// TIA Portal project "FactoryIO_Template_S7-1200_V16_V16" (V16)
// Vorlageprojekt für das Buch mit Zielsystem S7-1200

(* hardware
DEVICE "S7-1200-Station_1"  S7-1200 Station
   slot 0: "Baugruppenträger_0"  Rack  V1.0
   slot 1: "PLC_1"  CPU 1211C DC/DC/DC  6ES7 211-1AE40-0XB0  V4.1
*)

// ===== PLC "PLC_1"  CPU 1211C DC/DC/DC =====

VAR_GLOBAL   // PLC tag table "Standard-Variablentabelle"
   "belt_conv_0" AT %A0.0 : Bool;
   "start" AT %E0.0 : Bool;
   "stop" AT %E0.1 : Bool;
   "Tag_4" AT %I10.0 : Bool;
   "Tag_5" AT %Q10.0 : Bool;
   "Tag_6" AT %I10.1 : Bool;
   "run marker" AT %M0.0 : Bool;
   "stop load" AT %M0.4 : Bool;
   "Tag_3" AT %M6.1 : Bool;
   "belt_conv_0_Marker" AT %M5.0 : Bool;
   "Expect_off_Marker" AT %M1.7 : Bool;
   "run load" AT %M0.3 : Bool;
   "load_AC_marker" AT %M5.1 : Bool;
   "At_0_sens" AT %I0.5 : Bool;
   "mid_sens_Box" AT %I0.3 : Bool;
   "large_sens_Box" AT %I0.4 : Bool;
   "large_sens_marker" AT %M1.5 : Bool;
   "Tag_2" AT %M2.0 : Bool;
   "Expect_sens_marker" AT %M1.6 : Bool;
   "elevator_right_limit" AT %I1.2 : Bool;
   "Tag_7" AT %M0.2 : Bool;
   "Out_at_1_sens 11" AT %M1.0 : Bool;
   "At 2 High_sens _marker" AT %M2.4 : Bool;
   "Save_marker_Down" AT %M5.7 : Bool;
   "Save marker up" AT %M5.2 : Bool;
   "At_1_low_sens" AT %I0.6 : Bool;
   "Tag_8" AT %M0.5 : Bool;
   "out_at_1 sens" AT %M0.6 : Bool;
   "Slow_marker" AT %M5.3 : Bool;
   "At_low_sens_positive 2_marker" AT %M2.2 : Bool;
   "At_high_sens 1" AT %I0.7 : Bool;
   "Tag_9" AT %M0.7 : Bool;
   "Entry_1_Neg_marker" AT %M1.4 : Bool;
   "Entry_2_neg_marker" AT %M4.3 : Bool;
   "unload_marker" AT %M5.4 : Bool;
   "Entry_conv_1" AT %I1.3 : Bool;
   "Tag_10" AT %M1.1 : Bool;
   "entry_1_+_marker" AT %M1.2 : Bool;
   "Tag_11" AT %M1.3 : Bool;
   "belt_conv_1_marker" AT %M5.5 : Bool;
   "at_low_sens 2" AT %I1.0 : Bool;
   "Tag_12" AT %M2.1 : Bool;
   "at 2 high sens" AT %I1.1 : Bool;
   "Tag_13" AT %M2.3 : Bool;
   "entry_conv_2" AT %I1.4 : Bool;
   "Tag_14" AT %M4.2 : Bool;
   "Entry_2_+_marker" AT %M4.0 : Bool;
   "belt_conv_2_marker" AT %M5.6 : Bool;
   "load_Ac" AT %Q0.3 : Bool;
   "up" AT %Q0.5 : Bool;
   "slow" AT %Q0.7 : Bool;
   "unload" AT %Q0.4 : Bool;
   "belt_conv_1" AT %Q0.1 : Bool;
   "belt_conv_2" AT %Q0.2 : Bool;
   "down" AT %Q0.6 : Bool;
   "Tag_1" AT %M4.1 : Bool;
END_VAR

FUNCTION "MHJ-PLC-Lab-Function-S71200" : Void   // FC9000, SCL
{ S7_Optimized_Access := 'TRUE' }
VERSION : 0.1
   VAR_TEMP
      rdTimeReturn : Int;
      outputTime : DTL;
      SyncVal : Byte;
      forVal : Int;
      forVal_2 : Int;
      Value : Byte;
   END_VAR
   VAR CONSTANT
      CompVal : Byte := 16#34;
      Value_01 : Byte := 16#11;
      Value_01_DW : DWord := 16#A165_D992;
      Value_02_DW : DWord := 16#58BE_4401;
   END_VAR
BEGIN

   #Value:=PEEK(area := 16#82,
        dbNumber := 0,
        byteOffset := 511);
   #Value := #Value + 1;

   POKE(area := 16#82,
        dbNumber := 0,
        byteOffset := 511,
        value := #Value);

   POKE(area:=16#81,
        dbNumber:=0,
        byteOffset:=1016,
        value:=#Value_01_DW);
   POKE(area := 16#81,
        dbNumber := 0,
        byteOffset := 1020,
        value := #Value_02_DW);

   POKE(area := 16#81,
        dbNumber := 0,
        byteOffset := 511,
        value := B#16#00);

   FOR #forVal := 0 TO 120 DO
       FOR #forVal_2:=0 TO 10 DO
           #rdTimeReturn:=RD_SYS_T(#outputTime);
           #rdTimeReturn := WR_SYS_T(#outputTime);
           #rdTimeReturn := RD_SYS_T(#outputTime);
           #rdTimeReturn := WR_SYS_T(#outputTime);
       END_FOR;
       #SyncVal:= PEEK(area := 16#81,
                      dbNumber := 0,
                      byteOffset := 511);
       IF #SyncVal = #CompVal THEN
          GOTO M_1;
       END_IF;
   END_FOR;
   RETURN;

   M_1:
   POKE(area := 16#81,
        dbNumber := 0,
        byteOffset := 511,
        value := B#16#0);
END_FUNCTION

ORGANIZATION_BLOCK "Main"   // OB1, LAD, ProgramCycle
TITLE = "Main Program Sweep (Cycle)"
{ S7_Optimized_Access := 'TRUE' }
VERSION : 0.1
   VAR_INPUT
      Initial_Call : Bool;   // Initial call of this OB
      Remanence : Bool;   // =True, if remanent data are available
   END_VAR
   VAR_TEMP   // added for the SCL form of the ladder/FBD networks
      _w1 : Bool;
      _w2 : Bool;
      _w3 : Bool;
      _w4 : Bool;
      _w5 : Bool;
      _w6 : Bool;
      _w7 : Bool;
      _w8 : Bool;
      _w9 : Bool;
      _w10 : Bool;
   END_VAR
BEGIN

REGION Network 1: Konnektierungsbaustein für PLC-Lab
   // Im Netzwerk 1 wird der Konnektierungsbaustein für PLC-Lab aufgerufen.
   // Dieser Aufruf darf nicht entfernt werden!
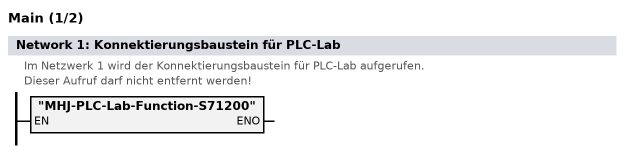
   RUNG wire#powerrail
      "MHJ-PLC-Lab-Function-S71200"()
   END_RUNG
   // the same network as SCL:
   "MHJ-PLC-Lab-Function-S71200"();
END_REGION

REGION Network 2
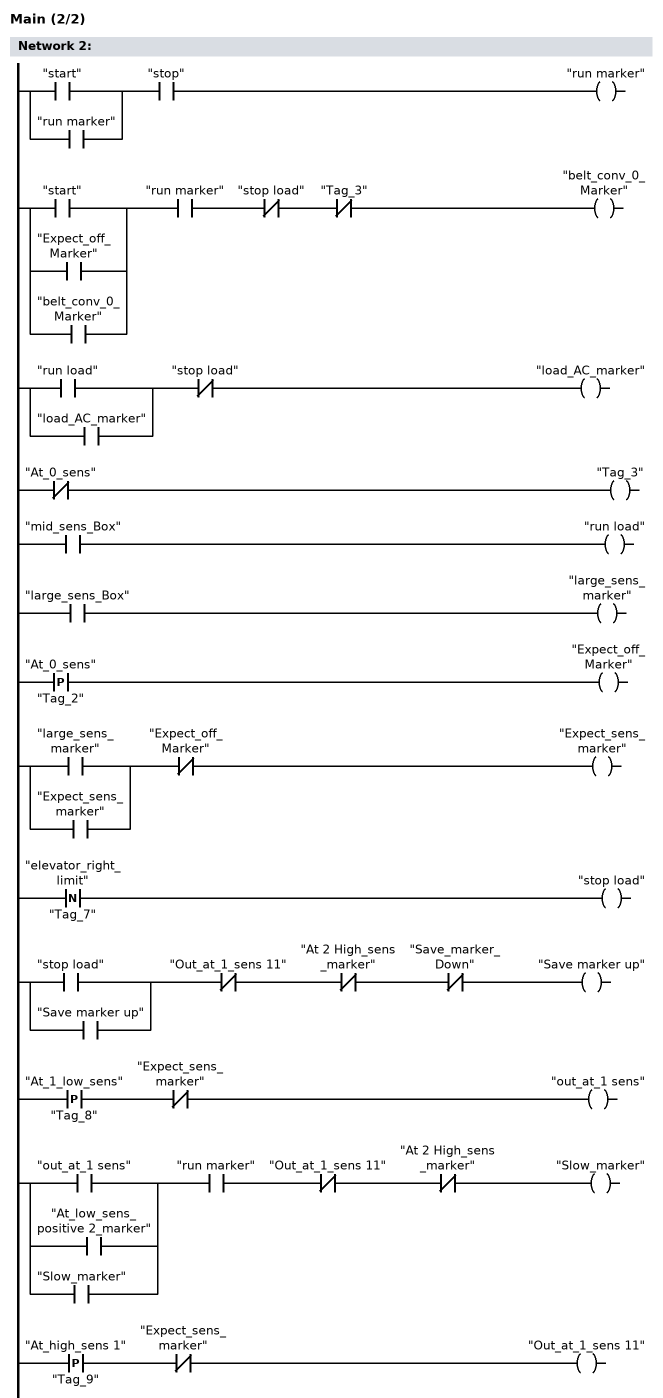
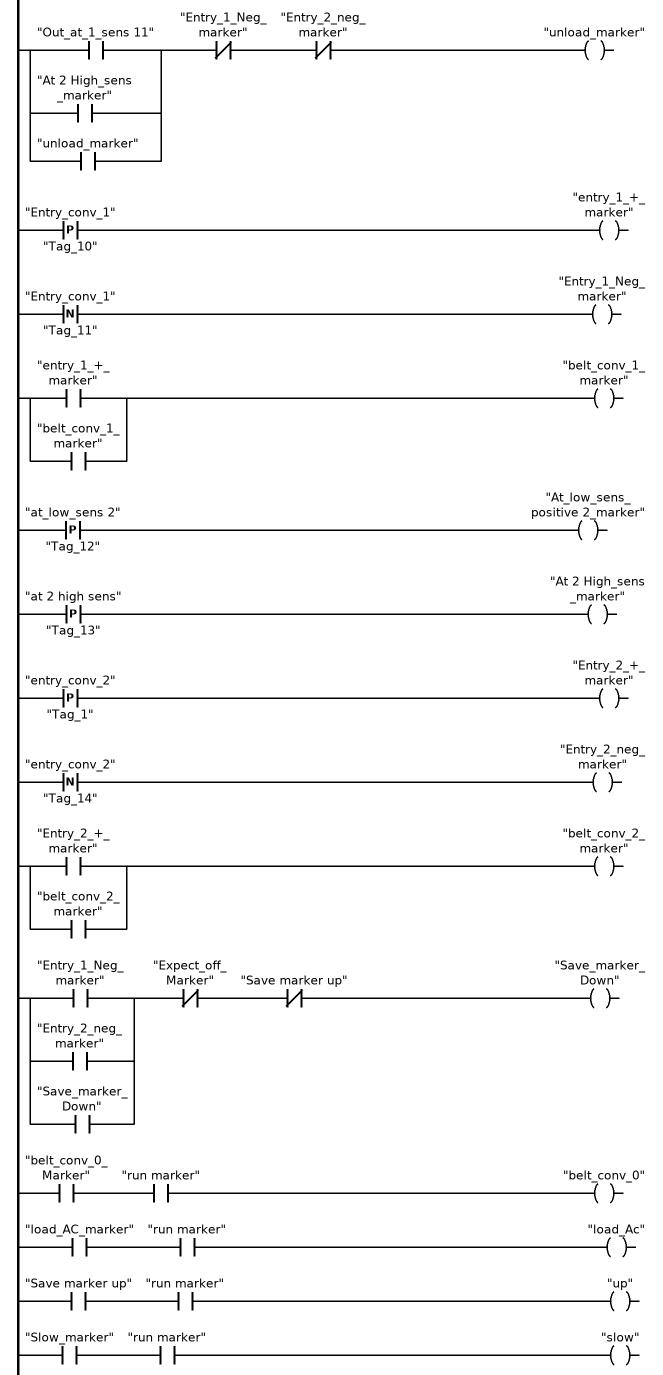
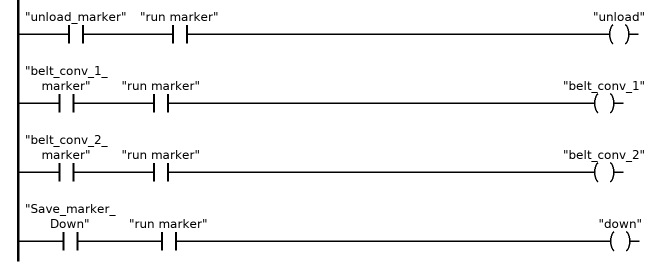
   RUNG wire#powerrail
      Contact( "start" )
      wire#w1
      Contact( "stop" )
      Coil( "run marker" )
   END_RUNG
   RUNG wire#powerrail
      Contact( "run marker" )
   END_RUNG wire#w1
   RUNG wire#powerrail
      Contact( "start" )
      wire#w2
      Contact( "run marker" )
      I_Contact( "stop load" )
      I_Contact( "Tag_3" )
      Coil( "belt_conv_0_Marker" )
   END_RUNG
   RUNG wire#powerrail
      Contact( "Expect_off_Marker" )
   END_RUNG wire#w2
   RUNG wire#powerrail
      Contact( "belt_conv_0_Marker" )
   END_RUNG wire#w2
   RUNG wire#powerrail
      Contact( "run load" )
      wire#w3
      I_Contact( "stop load" )
      Coil( "load_AC_marker" )
   END_RUNG
   RUNG wire#powerrail
      Contact( "load_AC_marker" )
   END_RUNG wire#w3
   RUNG wire#powerrail
      I_Contact( "At_0_sens" )
      Coil( "Tag_3" )
   END_RUNG
   RUNG wire#powerrail
      Contact( "mid_sens_Box" )
      Coil( "run load" )
   END_RUNG
   RUNG wire#powerrail
      Contact( "large_sens_Box" )
      Coil( "large_sens_marker" )
   END_RUNG
   RUNG wire#powerrail
      P_Contact(operand := "At_0_sens", bit := "Tag_2")
      Coil( "Expect_off_Marker" )
   END_RUNG
   RUNG wire#powerrail
      Contact( "large_sens_marker" )
      wire#w4
      I_Contact( "Expect_off_Marker" )
      Coil( "Expect_sens_marker" )
   END_RUNG
   RUNG wire#powerrail
      Contact( "Expect_sens_marker" )
   END_RUNG wire#w4
   RUNG wire#powerrail
      N_Contact(operand := "elevator_right_limit", bit := "Tag_7")
      Coil( "stop load" )
   END_RUNG
   RUNG wire#powerrail
      Contact( "stop load" )
      wire#w5
      I_Contact( "Out_at_1_sens 11" )
      I_Contact( "At 2 High_sens _marker" )
      I_Contact( "Save_marker_Down" )
      Coil( "Save marker up" )
   END_RUNG
   RUNG wire#powerrail
      Contact( "Save marker up" )
   END_RUNG wire#w5
   RUNG wire#powerrail
      P_Contact(operand := "At_1_low_sens", bit := "Tag_8")
      I_Contact( "Expect_sens_marker" )
      Coil( "out_at_1 sens" )
   END_RUNG
   RUNG wire#powerrail
      Contact( "out_at_1 sens" )
      wire#w6
      Contact( "run marker" )
      I_Contact( "Out_at_1_sens 11" )
      I_Contact( "At 2 High_sens _marker" )
      Coil( "Slow_marker" )
   END_RUNG
   RUNG wire#powerrail
      Contact( "At_low_sens_positive 2_marker" )
   END_RUNG wire#w6
   RUNG wire#powerrail
      Contact( "Slow_marker" )
   END_RUNG wire#w6
   RUNG wire#powerrail
      P_Contact(operand := "At_high_sens 1", bit := "Tag_9")
      I_Contact( "Expect_sens_marker" )
      Coil( "Out_at_1_sens 11" )
   END_RUNG
   RUNG wire#powerrail
      Contact( "Out_at_1_sens 11" )
      wire#w7
      I_Contact( "Entry_1_Neg_marker" )
      I_Contact( "Entry_2_neg_marker" )
      Coil( "unload_marker" )
   END_RUNG
   RUNG wire#powerrail
      Contact( "At 2 High_sens _marker" )
   END_RUNG wire#w7
   RUNG wire#powerrail
      Contact( "unload_marker" )
   END_RUNG wire#w7
   RUNG wire#powerrail
      P_Contact(operand := "Entry_conv_1", bit := "Tag_10")
      Coil( "entry_1_+_marker" )
   END_RUNG
   RUNG wire#powerrail
      N_Contact(operand := "Entry_conv_1", bit := "Tag_11")
      Coil( "Entry_1_Neg_marker" )
   END_RUNG
   RUNG wire#powerrail
      Contact( "entry_1_+_marker" )
      wire#w8
      Coil( "belt_conv_1_marker" )
   END_RUNG
   RUNG wire#powerrail
      Contact( "belt_conv_1_marker" )
   END_RUNG wire#w8
   RUNG wire#powerrail
      P_Contact(operand := "at_low_sens 2", bit := "Tag_12")
      Coil( "At_low_sens_positive 2_marker" )
   END_RUNG
   RUNG wire#powerrail
      P_Contact(operand := "at 2 high sens", bit := "Tag_13")
      Coil( "At 2 High_sens _marker" )
   END_RUNG
   RUNG wire#powerrail
      P_Contact(operand := "entry_conv_2", bit := "Tag_1")
      Coil( "Entry_2_+_marker" )
   END_RUNG
   RUNG wire#powerrail
      N_Contact(operand := "entry_conv_2", bit := "Tag_14")
      Coil( "Entry_2_neg_marker" )
   END_RUNG
   RUNG wire#powerrail
      Contact( "Entry_2_+_marker" )
      wire#w9
      Coil( "belt_conv_2_marker" )
   END_RUNG
   RUNG wire#powerrail
      Contact( "belt_conv_2_marker" )
   END_RUNG wire#w9
   RUNG wire#powerrail
      Contact( "Entry_1_Neg_marker" )
      wire#w10
      I_Contact( "Expect_off_Marker" )
      I_Contact( "Save marker up" )
      Coil( "Save_marker_Down" )
   END_RUNG
   RUNG wire#powerrail
      Contact( "Entry_2_neg_marker" )
   END_RUNG wire#w10
   RUNG wire#powerrail
      Contact( "Save_marker_Down" )
   END_RUNG wire#w10
   RUNG wire#powerrail
      Contact( "belt_conv_0_Marker" )
      Contact( "run marker" )
      Coil( "belt_conv_0" )
   END_RUNG
   RUNG wire#powerrail
      Contact( "load_AC_marker" )
      Contact( "run marker" )
      Coil( "load_Ac" )
   END_RUNG
   RUNG wire#powerrail
      Contact( "Save marker up" )
      Contact( "run marker" )
      Coil( "up" )
   END_RUNG
   RUNG wire#powerrail
      Contact( "Slow_marker" )
      Contact( "run marker" )
      Coil( "slow" )
   END_RUNG
   RUNG wire#powerrail
      Contact( "unload_marker" )
      Contact( "run marker" )
      Coil( "unload" )
   END_RUNG
   RUNG wire#powerrail
      Contact( "belt_conv_1_marker" )
      Contact( "run marker" )
      Coil( "belt_conv_1" )
   END_RUNG
   RUNG wire#powerrail
      Contact( "belt_conv_2_marker" )
      Contact( "run marker" )
      Coil( "belt_conv_2" )
   END_RUNG
   RUNG wire#powerrail
      Contact( "Save_marker_Down" )
      Contact( "run marker" )
      Coil( "down" )
   END_RUNG
   // the same network as SCL:
   "run marker" := ("start" OR "run marker") AND "stop";
   "belt_conv_0_Marker" := ("start" OR "Expect_off_Marker" OR "belt_conv_0_Marker") AND "run marker" AND NOT "stop load" AND NOT "Tag_3";
   "load_AC_marker" := ("run load" OR "load_AC_marker") AND NOT "stop load";
   "Tag_3" := NOT "At_0_sens";
   "run load" := "mid_sens_Box";
   "large_sens_marker" := "large_sens_Box";
   #_w1 := "At_0_sens" AND NOT "Tag_2";   // rising edge of "At_0_sens"
   "Tag_2" := "At_0_sens";
   "Expect_off_Marker" := #_w1;
   "Expect_sens_marker" := ("large_sens_marker" OR "Expect_sens_marker") AND NOT "Expect_off_Marker";
   #_w2 := NOT "elevator_right_limit" AND "Tag_7";   // falling edge of "elevator_right_limit"
   "Tag_7" := "elevator_right_limit";
   "stop load" := #_w2;
   "Save marker up" := ("stop load" OR "Save marker up") AND NOT "Out_at_1_sens 11" AND NOT "At 2 High_sens _marker" AND NOT "Save_marker_Down";
   #_w3 := "At_1_low_sens" AND NOT "Tag_8";   // rising edge of "At_1_low_sens"
   "Tag_8" := "At_1_low_sens";
   "out_at_1 sens" := #_w3 AND NOT "Expect_sens_marker";
   "Slow_marker" := ("out_at_1 sens" OR "At_low_sens_positive 2_marker" OR "Slow_marker") AND "run marker" AND NOT "Out_at_1_sens 11" AND NOT "At 2 High_sens _marker";
   #_w4 := "At_high_sens 1" AND NOT "Tag_9";   // rising edge of "At_high_sens 1"
   "Tag_9" := "At_high_sens 1";
   "Out_at_1_sens 11" := #_w4 AND NOT "Expect_sens_marker";
   "unload_marker" := ("Out_at_1_sens 11" OR "At 2 High_sens _marker" OR "unload_marker") AND NOT "Entry_1_Neg_marker" AND NOT "Entry_2_neg_marker";
   #_w5 := "Entry_conv_1" AND NOT "Tag_10";   // rising edge of "Entry_conv_1"
   "Tag_10" := "Entry_conv_1";
   "entry_1_+_marker" := #_w5;
   #_w6 := NOT "Entry_conv_1" AND "Tag_11";   // falling edge of "Entry_conv_1"
   "Tag_11" := "Entry_conv_1";
   "Entry_1_Neg_marker" := #_w6;
   "belt_conv_1_marker" := "entry_1_+_marker" OR "belt_conv_1_marker";
   #_w7 := "at_low_sens 2" AND NOT "Tag_12";   // rising edge of "at_low_sens 2"
   "Tag_12" := "at_low_sens 2";
   "At_low_sens_positive 2_marker" := #_w7;
   #_w8 := "at 2 high sens" AND NOT "Tag_13";   // rising edge of "at 2 high sens"
   "Tag_13" := "at 2 high sens";
   "At 2 High_sens _marker" := #_w8;
   #_w9 := "entry_conv_2" AND NOT "Tag_1";   // rising edge of "entry_conv_2"
   "Tag_1" := "entry_conv_2";
   "Entry_2_+_marker" := #_w9;
   #_w10 := NOT "entry_conv_2" AND "Tag_14";   // falling edge of "entry_conv_2"
   "Tag_14" := "entry_conv_2";
   "Entry_2_neg_marker" := #_w10;
   "belt_conv_2_marker" := "Entry_2_+_marker" OR "belt_conv_2_marker";
   "Save_marker_Down" := ("Entry_1_Neg_marker" OR "Entry_2_neg_marker" OR "Save_marker_Down") AND NOT "Expect_off_Marker" AND NOT "Save marker up";
   "belt_conv_0" := "belt_conv_0_Marker" AND "run marker";
   "load_Ac" := "load_AC_marker" AND "run marker";
   "up" := "Save marker up" AND "run marker";
   "slow" := "Slow_marker" AND "run marker";
   "unload" := "unload_marker" AND "run marker";
   "belt_conv_1" := "belt_conv_1_marker" AND "run marker";
   "belt_conv_2" := "belt_conv_2_marker" AND "run marker";
   "down" := "Save_marker_Down" AND "run marker";
END_REGION
END_ORGANIZATION_BLOCK